// Mitsubishi GX Works2 project: ch5   PLC: FX3U/FX3UC

PROGRAM MAIN
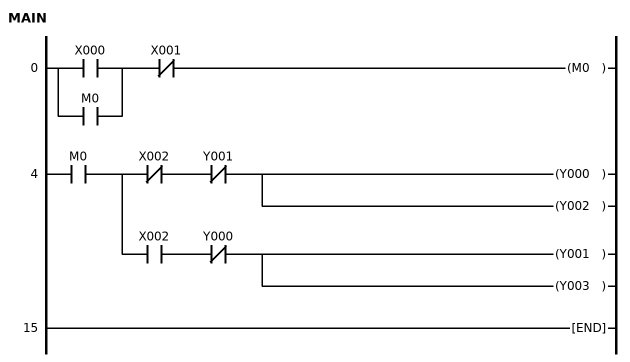
0     LD      X000
      OR      M0
      ANI     X001
      OUT     M0
4     LD      M0
      MPS
      ANI     X002
      ANI     Y001
      OUT     Y000
      OUT     Y002
      MPP
      AND     X002
      ANI     Y000
      OUT     Y001
      OUT     Y003
15    END
END_PROGRAM
